FUNCTION F_Current : REAL
VAR_INPUT
	I_Reading				: INT;
END_VAR
VAR
END_VAR

// Calvin - F_Current
// Rev 1.0 - April 6, 2023

F_Current					:= INT_TO_REAL(I_Reading) / 163.835;

END_FUNCTION

(* stored: Version 1.1.0.1, ProductVersion 3.1.4024.12
   POU F_Current: Id {7bbfe232-33e3-452f-b368-50ff52d822fe}, SpecialFunc None *)
